FUNCTION FC_LimitMinReal : bool
VAR_INPUT
	iMaster:	REAL;
END_VAR
VAR_IN_OUT
	ioSlave:		REAL;
END_VAR

IF (ioSlave < iMaster) THEN
	ioSlave := iMaster;
END_IF

END_FUNCTION

(* stored: Version 1.1.0.1, ProductVersion 3.1.4026.18
   POU FC_LimitMinReal: Id {0bad8ad8-4773-4985-8ba0-8d7c44224980}, SpecialFunc None *)
